PROGRAM MAIN
VAR
	
    fbStatusLight : FB_StatusLight;
    fbVereinzelung : FB_Vereinzelung;
    fbFoerderband : FB_Foerderband;
	fbDispenser1 : FB_Dispenser;
	fbDispenser2 : FB_Dispenser;
	fbDispenser3 : FB_Dispenser;

    bEnable : BOOL := FALSE;
    bExecute : BOOL := FALSE;
    nState_main : INT := 0;
    timer : TON;
	
	
END_VAR

// Zuweisung der globalen Variablen
bEnable := IFC_HW.bEnable;
bExecute := IFC_HW.bExecute;

// Initialisierung der Funktionsbausteine mit den globalen Variablen
fbStatusLight(eStatus := fbVereinzelung.eStatus, bRed => bAmpelRot, bYellow => bAmpelGelb, bGreen => bAmpelGrun);

fbVereinzelung(
    bSensor_1 := bEinzelSens1, 
    bSensor_2 := bEinzelSens2,
    bAkt1_1 => bR2AKT1,
    bAkt1_2 => bR1AKT1,
    bAkt2_1 => bR2AKT2,
    bAkt2_2 => bR1AKT2
);

fbFoerderband(
	bSensor1:= IFC_HW.bBandSens1, 
	bSensor2:= IFC_HW.bBandSens2, 
	bSensor3:= IFC_HW.bBandSens3, 
	bSensor4:= IFC_HW.bBandSens4, 
	ax :=  IFC_HW.ax_BandMotor, 
	bStopper1=> IFC_HW.bBandHub1, 
	bStopper2=> IFC_HW.bBandHub2, 
	bStopper3=> IFC_HW.bBandHub3
	);

fbDispenser1( 
    ax := IFC_HW.ax_Extruder1
);

fbDispenser2( 
    ax := IFC_HW.ax_Extruder2
);

fbDispenser3( 
    ax := IFC_HW.ax_Extruder3
);

fbDispenser1.nDispenceGram := 5;
fbDispenser2.nDispenceGram := 2;
fbDispenser3.nDispenceGram := 7;

IF NOT bEnable THEN
    nState_main := 0;
END_IF

CASE nState_main OF
    0:  // Off
        fbVereinzelung.bEnable := FALSE;
        fbFoerderband.bEnable := FALSE;
		fbDispenser1.bEnable := FALSE;
		fbDispenser2.bEnable := FALSE;
		fbDispenser3.bEnable := FALSE;

        IF bEnable THEN 
            nState_main := 1;
        END_IF

    1:  // Turn on
        fbVereinzelung.bEnable := TRUE;
  		fbFoerderband.bEnable := TRUE;
		fbDispenser1.bEnable := TRUE;
		fbDispenser2.bEnable := TRUE;
		fbDispenser3.bEnable := TRUE;

        IF fbVereinzelung.eStatus = State.Ready AND fbFoerderband.eStatus = State.Ready AND fbDispenser1.eStatus = State.Ready AND fbDispenser2.eStatus = State.Ready AND fbDispenser3.eStatus = State.Ready THEN
            nState_main := nState_main + 1;
        END_IF

    2:  // Vereinzeln
        IF bExecute THEN
            fbVereinzelung.bExecute := TRUE;
            IF fbVereinzelung.eStatus = State.Production THEN
                fbVereinzelung.bExecute := FALSE;
				nState_main := nState_main + 1;
            END_IF
        END_IF

	3:	// Fahre zu pos. 1
		fbFoerderband.bExecute := TRUE;		
		IF fbFoerderband.eStatus = State.Done THEN
			fbFoerderband.bExecute := FALSE;
			timer(in := TRUE, pt := T#2S);
			IF timer.q THEN
				timer.IN := FALSE;
				nState_main := nState_main + 1;
			END_IF 
		END_IF
		
	4: // Starte Dispenser 1
		fbDispenser1.bExecute := TRUE;
		IF fbDispenser1.bDone THEN
			fbDispenser1.bExecute := FALSE;
			nState_main := nState_main + 1;
		END_IF
		
	5: 	// fahre zu pos. 2
		fbFoerderband.bExecute := TRUE;
		IF fbFoerderband.eStatus = State.Done THEN
			fbFoerderband.bExecute := FALSE;
			timer(in := TRUE, pt := T#2S);
			IF timer.q THEN
				timer.IN := FALSE;
				nState_main := nState_main + 1;
			END_IF 
		END_IF
		
	6:	// Starte Dispenser 2
		fbFoerderband.bExecute := FALSE;
		fbDispenser2.bExecute := TRUE;
		IF fbDispenser2.eStatus = State.Done THEN
			fbDispenser2.bExecute := FALSE;
			nState_main := nState_main + 1;
		END_IF
		
	7: 	// fahre zu pos. 3
		fbFoerderband.bExecute := TRUE;
		IF fbFoerderband.eStatus = State.Done THEN
			fbFoerderband.bExecute := FALSE;
			nState_main := nState_main + 1;
		END_IF
		
	8:	// Starte Dispenser 3
		fbDispenser3.bExecute := TRUE;
		IF fbDispenser3.eStatus = State.Done THEN
			fbDispenser3.bExecute := FALSE;
			nState_main := nState_main + 1;
		END_IF
	
	9:	// fahre zu pos.4 
		fbFoerderband.bExecute := TRUE;
		IF fbFoerderband.eStatus = State.Done THEN
			fbFoerderband.bExecute := FALSE;
			nState_main := nState_main + 1;
		END_IF
	
		
		
		
		
		
		
		
		
		
		
		
		
		
		
		
		
END_CASE

END_PROGRAM

(* stored: Version 1.1.0.1, ProductVersion 3.1.4024.12
   POU MAIN: Id {41a6afe7-d655-4a0c-8495-2b17c7f15b36}, SpecialFunc None *)
